FUNCTION FinishAction 
VAR_INPUT
	StartAsync : BOOL := FALSE;
END_VAR
VAR
END_VAR

G_Match.bActionFinie := TRUE; //arrête l'action sans arrêter la partie asynchrone
IF NOT StartAsync THEN        //arrête l'action asynchrone
	G_Match.iAsyncAction := ''; 
	G_Match.iEtapeAction := 0;
END_IF

END_FUNCTION

(* stored: Version 1.1.0.1, ProductVersion 3.1.4024.12
   POU FinishAction: Id {64a2e075-7474-4a98-af0d-323ec0420576}, SpecialFunc None *)
